TYPE stCNTStatusCompact :
STRUCT
	{attribute addProperty Name "Bit 1(address x.0)"}
	Bit_1 : BIT;
	{attribute addProperty Name "Bit 2(address x.1)"}
	Bit_2 : BIT;
	{attribute addProperty Name "Set counter done"}
	SetCounterDone : BIT;
	{attribute addProperty Name "Counter inhibited"}
	CounterInhibited : BIT;
	{attribute addProperty Name "Bit 5(address x.4)"}
	Bit_5 : BIT;
	{attribute addProperty Name "Status of input clock"}
	StatusOfInputClock : BIT;
	{attribute addProperty Name "Bit 7(address x.6)"}
	Bit_7 : BIT;
	{attribute addProperty Name "Bit 8(address x.7)"}
	Bit_8 : BIT;
	{attribute addProperty Name "Bit 9(address x+1.0)"}
	Bit_9 : BIT;
	{attribute addProperty Name "Bit 10(address x+1.1)"}
	Bit_10 : BIT;
	{attribute addProperty Name "Bit 11(address x+1.2)"}
	Bit_11 : BIT;
	{attribute addProperty Name "Bit 12(address x+1.3)"}
	Bit_12 : BIT;
	{attribute addProperty Name "Bit 13(address x+1.4)"}
	Bit_13 : BIT;
	{attribute addProperty Name "Bit 14(address x+1.5)"}
	Bit_14 : BIT;
	{attribute addProperty Name "Bit 15(address x+1.6)"}
	Bit_15 : BIT;
	{attribute addProperty Name "TxPDO Toggle"}
	TxPDOToggle : BIT;
END_STRUCT
END_TYPE

(* stored: Version 1.1.0.1, ProductVersion 3.1.4024.9
   DUT stCNTStatusCompact: Id {42c8d20b-f917-0cbd-00b8-29ca7377d7e2} *)
